// TIA Portal project "1500Test" (V15)
// 2021-1-14 v1.0

(* hardware
DEVICE "S71500/ET200MP station_2"  S7-1500 station
   slot 0: "导轨_0"  Rack  6ES7 590-1***0-0AA0
   slot 1: "下"  CPU 1513-1 PN  6ES7 513-1AL02-0AB0  V2.5
      slot 3: "CPU 显示_1"  6ES7591-1AA00-0AA0
*)

// ===== PLC "下"  CPU 1513-1 PN =====

VAR_GLOBAL   // PLC tag table "默认变量表"
   "Tag_1" AT %I0.0 : "Type";
   "Tag_2" AT %Q0.0 : "Type";
   "Tag_4" AT %MB1 : Byte;
   "Tag_5" AT %MW2 : Word;
   "Tag_6" AT %MW4 : Int;
   "Tag_7" AT %MD6 : DWord;
   "Tag_8" AT %MD10 : DInt;
   "Tag_9" AT %MD14 : Real;
   "Tag_10" AT %M18.0 : LWord;
   "Tag_11" AT %M26.0 : LInt;
   "Tag_12" AT %M34.0 : LReal;
   "Clock_Byte" AT %MB0 : Byte;
   "Clock_10Hz" AT %M0.0 : Bool;
   "Clock_5Hz" AT %M0.1 : Bool;
   "Clock_2.5Hz" AT %M0.2 : Bool;
   "Clock_2Hz" AT %M0.3 : Bool;
   "Clock_1.25Hz" AT %M0.4 : Bool;
   "Clock_1Hz" AT %M0.5 : Bool;
   "Clock_0.625Hz" AT %M0.6 : Bool;
   "Clock_0.5Hz" AT %M0.7 : Bool;
   "Tag_3" AT %M100.0 : Bool;
   "Tag_13" AT %M100.1 : Bool;
END_VAR

TYPE "Type"
   STRUCT
      Element_1 : Bool;
      Element_2 : Byte;
      Element_3 : Word;
      Element_4 : Int;
      Element_5 : DWord;
      Element_6 : DInt;
      Element_7 : Real;
      Element_8 : LWord;
      Element_9 : LInt;
      Element_10 : LReal;
   END_STRUCT;
END_TYPE

DATA_BLOCK "AutoCoolingData"   // DB1
{ S7_Optimized_Access := 'FALSE' }
VERSION : 0.1
   VAR
      Cooling : Array[0..10] of Struct
         冷却清除标志 : Bool;
         Done : Bool;   // 冷却完成标志
         StartFlag : Bool;   // 冷却启动
         ResetOk : Bool;   // 复位完成
         Alarm : Bool;   // 冷却故障
         "Cooling Valve in" : Bool;   // 冷却阀门输出
         "Cooling Valce back" : Bool;   // 冷却阀门输出回
         "Start Signal" : Bool;   // 冷却信号运行输出
         StartOk : Bool;   // 冷却启动成功
         StatusCode : Int;   // 冷却状态码
         "Process Valve" : Real;   // 温度显示
         "Pass Valve" : Real;   // 冷却过充量
         冷却温度设定 : Real;
      END_STRUCT;
   END_VAR
BEGIN
END_DATA_BLOCK

DATA_BLOCK "AutoHeatingData"   // DB2
{ S7_Optimized_Access := 'FALSE' }
VERSION : 0.1
   VAR
      Heating : Array[0..11] of Struct
         加热清除标志 : Bool;
         Done : Bool;   // 加热完成标志
         "Process Valve" : Real;   // 温度显示
         "Pass Valve" : Real;   // 加热过充量
         "Lower Valve" : Real;   // 加热底限
         "Upper Valve" : Real;   // 加热报警值
         "Heating Start Delay" : DInt;   // 加热延时启动
         "Hold time" : Real;   // 加热时间设定
         锅重量 : Real;
         Mode : Int;
         加热温度设定 : Real;
         StartFlag : Bool;   // 加热启动
         ResetOk : Bool;   // 复位完成标志位
         Alarm : Bool;   // 加热故障
         "HeatingValve in" : Bool;   // 加热阀门输出
         StartOk : Bool;   // 加热成功标志位
         HeatingValveBack : Bool;   // 冷凝阀排放输出
         "Start signal" : Bool;   // 加热运行信号输出
         "Condensated wate valve" : Bool;   // 冷凝水排污阀
         "Hold time remainder" : Real;   // 加热剩余时间
         "Status CODE" : Int;   // 加热状态码
      END_STRUCT;
   END_VAR
BEGIN
END_DATA_BLOCK

DATA_BLOCK "AutoProcessData"   // DB3
{ S7_Optimized_Access := 'FALSE' }
VERSION : 0.1
   VAR
      Process : Array[0..20] of Struct
         Start : Bool;
         Stop : Bool;
         Drive : Bool;
      END_STRUCT;
      Static_1 : Array[0..1] of Byte;
   END_VAR
BEGIN
END_DATA_BLOCK

DATA_BLOCK "AutoStircontrolData"   // DB4
{ S7_Optimized_Access := 'FALSE' }
VERSION : 0.1
   VAR
      "Stic control" : Array[0..20] of Struct
         电机实际转速 : Int;
         搅拌清除标志 : Bool;
         变频器运行信号 : Bool;
         搅拌完成位 : Bool;
         转速设定 : Bool;
         变频器驱动信号输出 : Bool;
         搅拌报警 : Bool;
         搅拌启动成功 : Bool;
         搅拌启动 : Bool;
         复位完成位 : Bool;
         搅拌运行信号 : Bool;
         无搅拌运行标志位 : Bool;
         电机转速设定输出 : Int;
         电机转速设定 : Int;
         搅拌时间设定 : Real;
         搅拌Mode : Int;
         搅拌剩余时间 : Real;
         搅拌转速暂存 : Int;
         搅拌状态码 : Int;
      END_STRUCT;
   END_VAR
BEGIN
END_DATA_BLOCK

DATA_BLOCK "AutoWaitforData"   // DB5
{ S7_Optimized_Access := 'FALSE' }
VERSION : 0.1
   VAR
      Waitfor : Array[0..10] of Struct
         StartFlag : Bool;   // 启动
         Done : Bool;   // 等待完成
         ResetOk : Bool;   // 复位完成
         等待清除标志 : Bool;
         Alarm : Bool;   // 等待报警
         Startsignal : Bool;
         StartOk : Bool;
         等待实际值 : Real;
         Statuscode : Int;
      END_STRUCT;
   END_VAR
BEGIN
END_DATA_BLOCK

DATA_BLOCK "AutoWeight controlData"   // DB6
{ S7_Optimized_Access := 'FALSE' }
VERSION : 0.1
   VAR
      "Weight control" : Array[0..11] of Struct
         过冲量设定 : Real;
         过冲量报警量设定 : Real;
         过冲量报警时间设定 : DInt;
         投料量 : Real;
         投料清除标志 : Bool;
         Done : Bool;
         StartFlag : Bool;
         ResetOk : Bool;
         ValveDrive : Bool;
         投料报警 : Bool;
         投料运行信号 : Bool;
         StartOk : Bool;
         实际投料量 : Real;
         实际过冲量 : Real;
         StatusCode : Int;
      END_STRUCT;
   END_VAR
BEGIN
END_DATA_BLOCK

DATA_BLOCK "数据块_1"   // DB7
{ S7_Optimized_Access := 'FALSE' }
VERSION : 0.1
   VAR
      Static_1 : Array[0..10] of Struct
         Static_1 : Bool;
         Static_2 : Byte;
         Static_3 : Word;
         Static_4 : Int;
         Static_5 : DWord;
         Static_6 : DInt;
         Static_7 : Real;
         Static_8 : LWord;
         Static_9 : LInt;
         Static_10 : LReal;
      END_STRUCT;
   END_VAR
BEGIN
END_DATA_BLOCK

DATA_BLOCK "数据块_2"   // DB8
{ S7_Optimized_Access := 'FALSE' }
VERSION : 0.1
   VAR
      Static_1 : Array[0..10] of Struct
         Static_1 : Bool;
         Static_2 : Byte;
         Static_3 : Word;
         Static_4 : Int;
         Static_5 : DWord;
         Static_6 : DInt;
         Static_7 : Real;
         Static_8 : LWord;
         Static_9 : LInt;
         Static_10 : LReal;
      END_STRUCT;
   END_VAR
BEGIN
END_DATA_BLOCK

DATA_BLOCK "数据块_3"   // DB9
{ S7_Optimized_Access := 'FALSE' }
VERSION : 0.1
   VAR
      Static_63 : Array[0..5] of Struct
         Static_1 : Bool;
         Static_2 : Byte;
         Static_3 : Word;
         Static_4 : Bool;
         Static_5 : Bool;
         Static_6 : Bool;
         Static_7 : Byte;
         Static_8 : Int;
         Static_9 : Word;
         Static_10 : DInt;
         Static_11 : DWord;
         Static_12 : DInt;
         Static_13 : Word;
         Static_14 : DWord;
         Static_15 : Real;
         Static_16 : LReal;
         Static_17 : LInt;
         Static_18 : LWord;
         Static_19 : Word;
         Static_20 : LInt;
         Static_21 : Bool;
         Static_22 : Bool;
         Static_23 : Bool;
         Static_24 : Bool;
         Static_25 : Bool;
         Static_26 : Bool;
         Static_27 : Bool;
         Static_28 : Bool;
         Static_29 : Bool;
         Static_30 : Bool;
         Static_31 : Bool;
         Static_32 : LInt;
         Static_33 : LReal;
         Static_34 : Byte;
         Static_35 : Int;
         Static_36 : Word;
         Static_37 : DInt;
         Static_38 : DWord;
         Static_39 : LReal;
         Static_40 : Real;
         Static_41 : Byte;
         Static_42 : Word;
         Static_43 : Bool;
         Static_44 : Bool;
         Static_45 : Bool;
         Static_46 : Bool;
         Static_47 : Bool;
         Static_48 : Bool;
         Static_49 : Bool;
         Static_50 : Bool;
         Static_51 : Bool;
         Static_52 : Word;
         Static_53 : DWord;
         Static_54 : DInt;
         Static_55 : DInt;
         Static_56 : DWord;
         Static_57 : DWord;
         Static_58 : Int;
         Static_59 : Byte;
         Static_60 : Byte;
         Static_61 : Byte;
         Static_62 : Byte;
      END_STRUCT;
   END_VAR
BEGIN
END_DATA_BLOCK

DATA_BLOCK "数据块_4"   // DB10
{ S7_Optimized_Access := 'FALSE' }
VERSION : 0.1
   VAR
      Static_1 : Array[0..10] of Bool;
      Static_2 : Array[0..10] of Byte;
      Static_3 : Array[0..10] of Int;
      Static_4 : Array[0..10] of Word;
      Static_5 : Array[0..10] of DInt;
      Static_6 : Array[0..10] of DWord;
      Static_7 : Array[0..10] of Real;
      Static_8 : Array[0..10] of LReal;
      Static_9 : Array[0..10] of LInt;
      Static_10 : Array[0..10] of LWord;
   END_VAR
BEGIN
END_DATA_BLOCK

DATA_BLOCK "数据块_5"   // DB11
{ S7_Optimized_Access := 'FALSE' }
VERSION : 0.1
   VAR
      Static_1 : Array[0..500] of Byte;
   END_VAR
BEGIN
END_DATA_BLOCK

DATA_BLOCK "数据块_6"   // DB12
{ S7_Optimized_Access := 'FALSE' }
VERSION : 0.1
   VAR
      Static_1 : Array[0..400] of Int;
   END_VAR
BEGIN
END_DATA_BLOCK

DATA_BLOCK "数据块_7"   // DB13
{ S7_Optimized_Access := 'FALSE' }
VERSION : 0.1
   VAR
      Static_1 : Array[0..400] of Word;
   END_VAR
BEGIN
END_DATA_BLOCK

DATA_BLOCK "数据块_8"   // DB14
{ S7_Optimized_Access := 'FALSE' }
VERSION : 0.1
   VAR
      Static_1 : Array[0..6000] of Bool;
   END_VAR
BEGIN
END_DATA_BLOCK

DATA_BLOCK "数据块_9"   // DB15
{ S7_Optimized_Access := 'FALSE' }
VERSION : 0.1
   VAR
      Static_1 : Array[0..200] of DInt;
   END_VAR
BEGIN
END_DATA_BLOCK

DATA_BLOCK "数据块_10"   // DB16
{ S7_Optimized_Access := 'FALSE' }
VERSION : 0.1
   VAR
      Static_1 : Array[0..200] of DWord;
   END_VAR
BEGIN
END_DATA_BLOCK

DATA_BLOCK "数据块_11"   // DB17
{ S7_Optimized_Access := 'FALSE' }
VERSION : 0.1
   VAR
      Static_1 : Array[0..200] of Real;
   END_VAR
BEGIN
END_DATA_BLOCK

DATA_BLOCK "数据块_12"   // DB18
{ S7_Optimized_Access := 'FALSE' }
VERSION : 0.1
   VAR
      Static_1 : Array[0..100] of LInt;
   END_VAR
BEGIN
END_DATA_BLOCK

DATA_BLOCK "数据块_13"   // DB19
{ S7_Optimized_Access := 'FALSE' }
VERSION : 0.1
   VAR
      Static_1 : Array[0..100] of LWord;
   END_VAR
BEGIN
END_DATA_BLOCK

DATA_BLOCK "数据块_14"   // DB20
{ S7_Optimized_Access := 'FALSE' }
VERSION : 0.1
   VAR
      Static_1 : Array[0..100] of LReal;
   END_VAR
BEGIN
END_DATA_BLOCK

FUNCTION "块_1" : Void   // FC1, SCL
{ S7_Optimized_Access := 'TRUE' }
VERSION : 0.1
   VAR_TEMP
      i : Int;
   END_VAR
BEGIN
   "数据块_5".Static_1[0] := 1 + "数据块_5".Static_1[0];
   FOR #i := 0 TO 500 DO
       "数据块_5".Static_1[#i] := "数据块_5".Static_1[0];;
   END_FOR;
   "数据块_6".Static_1[0] := 1 + "数据块_6".Static_1[0];
   #i := 0;
   FOR #i := 0 TO 400 DO

       "数据块_6".Static_1[#i] := "数据块_6".Static_1[0];
       ;
   END_FOR;

   "数据块_7".Static_1[0] := 1 + "数据块_7".Static_1[0];
   #i := 0;
   FOR #i := 0 TO 400 DO

       "数据块_7".Static_1[#i] := "数据块_7".Static_1[0];
       ;
   END_FOR;
   "数据块_8".Static_1[0] := NOT "数据块_8".Static_1[0];
   #i := 0;
   FOR #i := 0 TO 6000 DO

       "数据块_8".Static_1[#i] := "数据块_8".Static_1[0];
       ;
   END_FOR;

   "数据块_9".Static_1[0] :="数据块_9".Static_1[0]+1;
   #i := 0;
   FOR #i := 0 TO 200 DO

       "数据块_9".Static_1[#i] := "数据块_9".Static_1[0];
       ;
   END_FOR;

   "数据块_10".Static_1[0] := "数据块_10".Static_1[0] + 1;
   #i := 0;
   FOR #i := 0 TO 200 DO

       "数据块_10".Static_1[#i] := "数据块_10".Static_1[0];
       ;
   END_FOR;

   "数据块_11".Static_1[0] := "数据块_11".Static_1[0] + 1.0;
   #i := 0;
   FOR #i := 0 TO 200 DO

       "数据块_11".Static_1[#i] := "数据块_11".Static_1[0];
       ;
   END_FOR;

   "数据块_12".Static_1[0] := "数据块_12".Static_1[0] + 1;
   #i := 0;
   FOR #i := 0 TO 100 DO

       "数据块_12".Static_1[#i] := "数据块_12".Static_1[0];
       ;
   END_FOR;

   "数据块_13".Static_1[0] := "数据块_13".Static_1[0] + 1;
   #i := 0;
   FOR #i := 0 TO 100 DO

       "数据块_13".Static_1[#i] := "数据块_13".Static_1[0];
       ;
   END_FOR;

   "数据块_14".Static_1[0] := "数据块_14".Static_1[0] + 1.0;
   #i := 0;
   FOR #i := 0 TO 100 DO

       "数据块_14".Static_1[#i] := "数据块_14".Static_1[0];
       ;
   END_FOR;
END_FUNCTION

ORGANIZATION_BLOCK "Main"   // OB1, LAD, ProgramCycle
TITLE = "Main Program Sweep (Cycle)"
{ S7_Optimized_Access := 'TRUE' }
VERSION : 0.1
   VAR_INPUT
      Initial_Call : Bool;   // Initial call of this OB
      Remanence : Bool;   // =True, if remanent data are available
   END_VAR
   VAR_TEMP   // added for the SCL form of the ladder/FBD networks
      _w1 : Bool;
   END_VAR
BEGIN

REGION Network 1
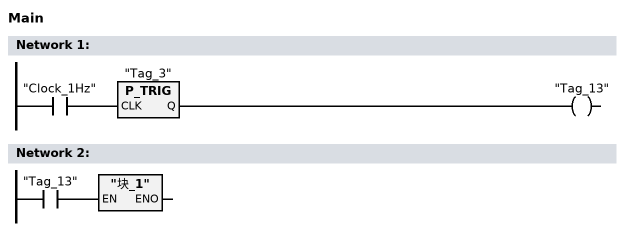
   RUNG wire#powerrail
      Contact( "Clock_1Hz" )
      P_Trig( "Tag_3" )
      Coil( "Tag_13" )
   END_RUNG
   // the same network as SCL:
   #_w1 := "Clock_1Hz" AND NOT "Tag_3";   // rising edge
   "Tag_3" := "Clock_1Hz";
   "Tag_13" := #_w1;
END_REGION

REGION Network 2
   RUNG wire#powerrail
      Contact( "Tag_13" )
      "块_1"()
   END_RUNG
   // the same network as SCL:
   IF "Tag_13" THEN "块_1"(); END_IF;
END_REGION
END_ORGANIZATION_BLOCK